(* Logix 5000 project; controller PID_Tanque Emulate 5570 rev 33.11; software revision 33.00 *)

TASK T00_MainTask (continuous, watchdog 500 ms) : P00_MainProgram

MODULES
   Local : Emulate 5570 (ICP 2, rev 33.11)
END_MODULES

VAR_GLOBAL   (* controller tags *)
   B00 : BOOL; {access None}   // Bandera Start
   INB_BT1 : BOOL;   // Boton Start
   INB_BT2 : BOOL;   // Boton Reset
   INB_BT3 : BOOL;   // Boton Stop
   INF_TFM : REAL;   // Sensor de Caudal
   INF_TLM : REAL;   // Sensor de nivel 0-10
   OUB_LB1 : BOOL;   // Boton Start
   OUB_LB2 : BOOL;   // Boton Reset
   OUB_LB3 : BOOL;   // Boton Stop
   OUF_TDV : REAL;   // Valvula de descarga
   OUF_TFV : REAL;   // Valvula de llenado
   TDV : REAL; {access None}   // DESCARGA
   TFV : REAL; {access None}   // Llenado de tanque
   TLM : REAL; {access None}   // Entrada escalada de sensor de nivel: 0-300
END_VAR

PROGRAM P00_MainProgram   (* main routine R00_MainRoutine *)
VAR
   Error : REAL;
   PID_Level : PID := (CTL := 33554432, CA := 1, KP := 1.6, KI := 0.2, KD := 0.1, MAXS := 300.0, MAXO := 100.0, UPD := 0.05, MAXI := 300.0, MAXCV := 100.0); {access None}   // Instruccion PID para control de nivel de tanque
   SCL_01 : SCALE; {access None}
END_VAR

ROUTINE R00_MainRoutine   (* ladder *)
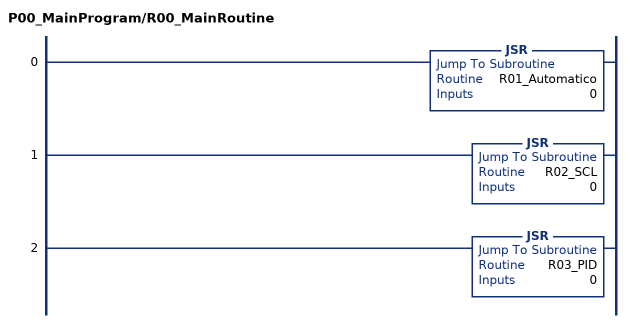
   0: JSR(R01_Automatico,0);
   1: JSR(R02_SCL,0);
   2: JSR(R03_PID,0);
END_ROUTINE

ROUTINE R01_Automatico   (* ladder *)
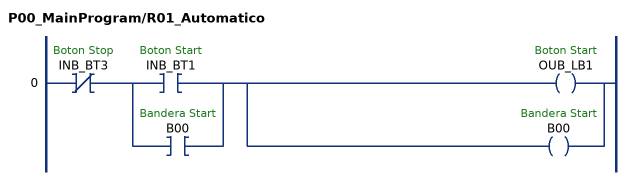
   0: XIO(INB_BT3)[XIC(INB_BT1) ,XIC(B00) ][OTE(OUB_LB1) ,OTE(B00) ];
END_ROUTINE

ROUTINE R02_SCL   (* function block diagram *)
   SHEET 1
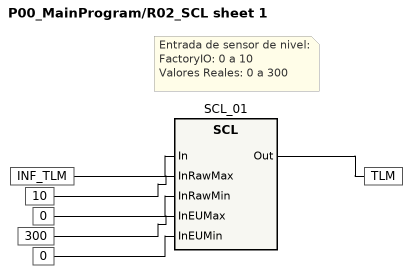
   // Entrada de sensor de nivel:
   // FactoryIO: 0 a 10
   // Valores Reales: 0 a 300
   SCL_01 : SCL(In := INF_TLM, InRawMax := 10, InRawMin := 0, InEUMax := 300, InEUMin := 0);
   TLM := SCL_01.Out;
END_ROUTINE

ROUTINE R03_PID   (* ladder *)
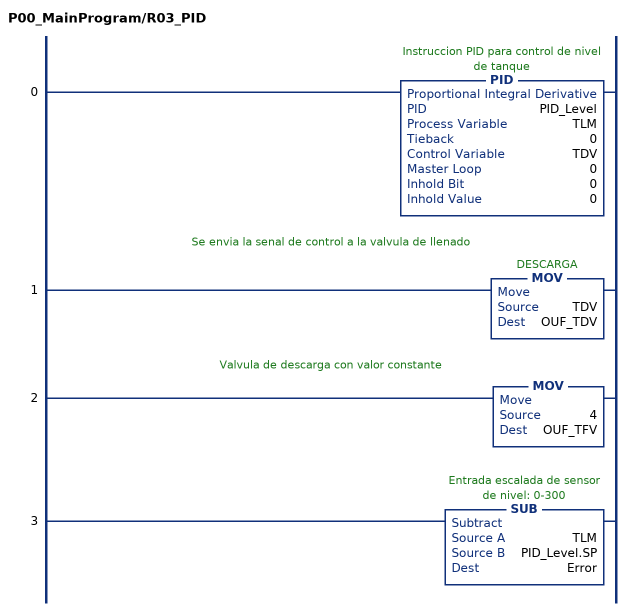
   0: PID(PID_Level,TLM,0,TDV,0,0,0);
   // Se envia la senal de control a la valvula de llenado
   1: MOV(TDV,OUF_TDV);
   // Valvula de descarga con valor constante
   2: MOV(4,OUF_TFV);
   3: SUB(TLM,PID_Level.SP,Error);
END_ROUTINE
END_PROGRAM
